// TwinCAT 3 PLC project PLC1
// ProgramVersion: 3.1.4026.22
// libraries:
//   Tc2_MC2, * (Beckhoff Automation GmbH)
//   Tc2_Standard, * (Beckhoff Automation GmbH)
//   Tc2_System, * (Beckhoff Automation GmbH)
//   Tc3_Mc3PlanarMotion, * (Beckhoff Automation GmbH)
//   Tc3_Physics, * (Beckhoff Automation GmbH)
//   Tc3_XPlanarUtility, * (Beckhoff Automation GmbH)
//   XPlanarApplication, * (Beckhoff Automation LLC)
// project tree:
//   GVLs/ GVL.TcGVL
//   / PlcTask.TcTTO
//   POUs/ MAIN.TcPOU
//   POUs/Utilities/ ErrorStep.TcPOU, NextMinorStep.TcPOU (not stored), NextStep.TcPOU (not stored)
//   POUs/XPlanarModule/ FB_XPlanarModule.TcPOU
//   POUs/XPlanarModule/StationProcesses/ FB_RotateStation.TcPOU, FB_SimulateProcess.TcPOU
// real-time tasks:
//   TASK XPlanar Task_3: cycle T#250us, priority 1, ADS port 350
//   TASK Job Task: cycle default, priority 2
//   TASK MC-Task (MET): cycle T#2ms, priority 3, ADS port 351
//   TASK MC-Task (MPT): cycle T#10ms, priority 4, ADS port 352
//   TASK PlcTask: cycle T#10ms, priority 20, ADS port 353
// variable links:
//   XPlanar MC Project/Axes/Mover4220_1 <-> TcCOM Objects/XPlanar/Mover4220_1
//     IoToMc/STD <-> OutputsToNC3/HWToNC3
//     McToIo/STD <-> InputsFromNC3/NC3ToHW
//   XPlanar MC Project/Axes/Mover4220_2 <-> TcCOM Objects/XPlanar/Mover4220_2
//     IoToMc/STD <-> OutputsToNC3/HWToNC3
//     McToIo/STD <-> InputsFromNC3/NC3ToHW
//   PLC1/PLC1 Instance <-> XPlanar MC Project/Axes/Mover4220_1
//     PlcTask Inputs/MAIN.XPlanarTable.Movers[1]._Mover.MCTOPLC/ACT <-> McToPlc/ACT
//     PlcTask Inputs/MAIN.XPlanarTable.Movers[1]._Mover.MCTOPLC/COORDMODE <-> McToPlc/COORDMODE
//     PlcTask Inputs/MAIN.XPlanarTable.Movers[1]._Mover.MCTOPLC/SET <-> McToPlc/SET
//     PlcTask Inputs/MAIN.XPlanarTable.Movers[1]._Mover.MCTOPLC/SETONTRACK <-> McToPlc/SETONTRACK
//     PlcTask Inputs/MAIN.XPlanarTable.Movers[1]._Mover.MCTOPLC/STD <-> McToPlc/STD
//     PlcTask Outputs/MAIN.XPlanarTable.Movers[1]._Mover.PLCTOMC/STD <-> PlcToMc/STD
//   PLC1/PLC1 Instance <-> XPlanar MC Project/Axes/Mover4220_2
//     PlcTask Inputs/MAIN.XPlanarTable.Movers[2]._Mover.MCTOPLC/ACT <-> McToPlc/ACT
//     PlcTask Inputs/MAIN.XPlanarTable.Movers[2]._Mover.MCTOPLC/COORDMODE <-> McToPlc/COORDMODE
//     PlcTask Inputs/MAIN.XPlanarTable.Movers[2]._Mover.MCTOPLC/SET <-> McToPlc/SET
//     PlcTask Inputs/MAIN.XPlanarTable.Movers[2]._Mover.MCTOPLC/SETONTRACK <-> McToPlc/SETONTRACK
//     PlcTask Inputs/MAIN.XPlanarTable.Movers[2]._Mover.MCTOPLC/STD <-> McToPlc/STD
//     PlcTask Outputs/MAIN.XPlanarTable.Movers[2]._Mover.PLCTOMC/STD <-> PlcToMc/STD
//   PLC1/PLC1 Instance <-> XPlanar MC Project/Groups/Environment
//     PlcTask Inputs/XPlanar.Environment.MCTOPLC_STD <-> McToPlc/STD
//   PLC1/PLC1 Instance <-> XPlanar MC Project/Groups/Track1
//     PlcTask Inputs/MAIN.XPlanarTable.Tracks[1]._Track.MCTOPLC_STD <-> McToPlc/STD
//   PLC1/PLC1 Instance <-> XPlanar MC Project/Groups/Track2
//     PlcTask Inputs/MAIN.XPlanarTable.Tracks[2]._Track.MCTOPLC_STD <-> McToPlc/STD
//   PLC1/PLC1 Instance <-> XPlanar MC Project/Groups/XPlanar
//     PlcTask Inputs/XPlanar.Group.MCTOPLC_STD <-> McToPlc/STD

CONFIGURATION PLC1
    RESOURCE PLC ON TwinCAT3
        TASK PlcTask(INTERVAL := T#10ms, PRIORITY := 20);
        PROGRAM MAIN WITH PlcTask : MAIN;
    END_RESOURCE
END_CONFIGURATION

// ---- GVLs/GVL.TcGVL
{attribute 'qualified_only'}
VAR_GLOBAL
	// Mover Velocity
	MoverVelo		: LREAL := 200;
	MoverGap		: LREAL := 180; // Do not exceed 250 mm, or go lower then default
	// Mover Rotation Velocity
	MoverSpinVelo	: LREAL := 1000;
	// Station 2 Mover Index
	Indx			: UDINT;
END_VAR

// ---- POUs/MAIN.TcPOU
PROGRAM MAIN
VAR
	XPlanarTable : FB_XPlanarModule;
	Initialize	 : BOOL; // Initialize the system
	Reset		 : BOOL; // Reset and Execute System
	Start		 : BOOL; // Run the system
	Halt		 : BOOL; // Avoid Disabling while spinning, otherwise physical sqauring of mover is required
	MachineState : (Startup,
		InitSystem,
		ResetSystem,
		Recover,
		Ready,
		Run,
		Disable);
	trig : R_TRIG;
END_VAR

//This project is a very simple "hello world" example for the APS4322 2-Tile starter kit.
//It is currently based on the XPlanarApplication library version 2.0.5 or greater.


//Keep all XPlanar motion system objects up to date every cycle
XPlanarTable.CyclicLogic();

// "Machine" Sequence
CASE MachineState OF
	Startup:	
		IF Initialize THEN
			Initialize := FALSE;
			MachineState := InitSystem;
		END_IF
	
	InitSystem:	
		IF XPlanarTable.Initialize() THEN
			MachineState := ResetSystem;
		END_IF
	
	ResetSystem:	
		IF Reset AND_THEN XPlanarTable.Reset() THEN
			Reset := FALSE;
			MachineState := Recover;
		END_IF
	
	Recover:	
		IF XPlanarTable.Recovery() THEN
			MachineState := Ready;
		END_IF
		
	Ready:
		IF Start THEN
			MachineState := Run;
		END_IF
	
	Run: 
		XPlanarTable.Execute();
	
	Disable:	
		IF XPlanarTable.Disable() THEN
			MachineState := 0;
		END_IF
END_CASE

IF Halt OR trig.Q THEN
	MachineState := Disable;
	Halt := FALSE;
END_IF

END_PROGRAM

// ---- POUs/XPlanarModule/FB_XPlanarModule.TcPOU
FUNCTION_BLOCK FB_XPlanarModule
VAR CONSTANT
	MoverCount	 : UDINT := 2;
	TrackCount	 : UDINT := 2;
	StationCount : UDINT := 2;
END_VAR

VAR
	XPlanarSystem	: FB_Component_XPlanar;
	Movers			: ARRAY[1..MoverCount] OF FB_XPlanarMover;
	Tracks			: ARRAY[1..TrackCount] OF FB_XPlanarTrackSegment;
	Stations		: ARRAY[1..StationCount] OF FB_XPlanarStationBase;
	Station1Process : FB_SimulateProcess;  //Custom process FB that can be assigned to a station
	Station2Process : FB_RotateStation;
	InitState		: (CheckForXPlanarInit, UpdateDynamics, SetStationParameters, Initialized);
END_VAR

METHOD CyclicLogic : BOOL
VAR
	i : UDINT;
END_VAR
VAR_INST
	TaskResult	: I_PlanarTaskResult;
END_VAR
XPlanarSystem.CyclicLogic();
IF NOT XPlanarSystem.Initialized THEN
	RETURN;
END_IF

//Add any logic that needs to be called every cycle here
END_METHOD

METHOD Disable : BOOL
VAR_INST
	CommandResult	: I_PlanarTaskResult;
END_VAR
CommandResult := XPlanarSystem.Abort(); // Stop Motion and Disable All Movers
IF CommandResult.Done THEN
	Disable := TRUE;
END_IF
END_METHOD

METHOD Execute : BOOL
VAR
	i : UDINT;
END_VAR
//System is 'running' cycle thru all of the stations
FOR i := 1 TO XPlanar.StationCount DO
	ip.Stations[i].Execute();
END_FOR
END_METHOD

METHOD Initialize : BOOL
VAR_INST
	i			: UDINT;
END_VAR
CASE InitState OF
	CheckForXPlanarInit: // Init Vars
		Initialize := FALSE;
		
		//Make sure the XPlanar motion system has initialized
		IF XPlanarSystem.Initialized THEN
			InitState := UpdateDynamics;
		END_IF

	UpdateDynamics: 
		//Assign Initial Application Mover Dynamics
		FOR i := 1 TO XPlanar.MoverCount DO
			ip.Movers[i].Gap						:= 200;
			ip.Movers[i].Dynamics.Movement.Velocity := GVL.MoverVelo;
			ip.Movers[i].Dynamics.Movement.Accel	:= GVL.MoverVelo * 10;
			ip.Movers[i].Dynamics.Movement.Decel	:= GVL.MoverVelo * 10;
			ip.Movers[i].Dynamics.Movement.Jerk		:= GVL.MoverVelo * 100;
			ip.Movers[i].Dynamics.Rotation.Velocity := GVL.MoverSpinVelo;
			ip.Movers[i].Dynamics.Rotation.Accel	:= GVL.MoverSpinVelo * 10;
			ip.Movers[i].Dynamics.Rotation.Decel	:= GVL.MoverSpinVelo * 10;
			ip.Movers[i].Dynamics.Rotation.Jerk		:= GVL.MoverSpinVelo * 100;
		END_FOR

		InitState := SetStationParameters;

	SetStationParameters:
		IF SetupStations() THEN
			InitState := Initialized;
		END_IF

	Initialized: // Init Complete
		Initialize := TRUE;
END_CASE
END_METHOD

METHOD Recovery : BOOL
VAR_INST
	nState			: UDINT;
	ipResult		: ARRAY[1..MoverCount] OF I_PlanarTaskResult;
	ErrorMoverId, i : UDINT;
	ItemsOk			: BOOL;
END_VAR
//This is an example of some very simple mover recovery.  
//What needs to be done to recover will be unique for each application.

CASE nState OF
	0: // Init Vars
		Recovery := FALSE;
		i := 1;
		NextStep(nState);
		
	10: // All Movers Join rack closest to their current location
		IF i <= XPlanar.MoverCount THEN
			ipResult[i] := ip.Movers[i].MoveCommand.JoinClosestTrack(FALSE);
			IF ipResult[i].Done THEN
				NextMinorStep(nState);
			ELSIF ipResult[i].Error THEN
				ErrorStep(nState);
			END_IF
		ELSE
			i := 1;
			NextStep(nState);
		END_IF

	11: //Check Mover Count
		IF i <= XPlanar.MoverCount THEN
			i	   := i + 1;
			nState := 10;
		ELSE
			i := 1;
			NextStep(nState);
		END_IF

	20: // Sort and send Movers to Stations
		FOR i := 1 TO XPlanar.MoverCount DO
			ipResult[i] := ip.Movers[i].MoveCommand.SendToStation(ip.Stations[1]);
		END_FOR

		NextStep(nState);

	30: // Wait For Mover to Move
		ItemsOk := TRUE;
		FOR i := 1 TO XPlanar.MoverCount DO
			IF NOT ipResult[i].Busy THEN
				ItemsOk := FALSE;
			END_IF

			IF ipResult[i].Error THEN
				ErrorMoverId := i;
				ErrorStep(nState);
			END_IF
		END_FOR

		IF ItemsOk THEN
			ErrorMoverId := 0;
			NextStep(nState);
		END_IF

	40: // Complete
		nState		 := 0;
		ErrorMoverId := 0;
		Recovery	 := TRUE;
END_CASE
END_METHOD

METHOD Reset : BOOL
VAR_INST
	nState		  : UDINT;
	i			  : UDINT;
	ResetOk		  : BOOL;
	ResetError	  : BOOL;
	CommandResult : I_PlanarTaskResult;
END_VAR
CASE nState OF
	0: // Init Vars
		Reset := FALSE;
		NextStep(nState);

	10: // Reset Table 
		IF XPlanarSystem.Reset().Done THEN
			NextStep(nState);
		END_IF

	20: // Reset Stations
		FOR i := 1 TO StationCount DO
			ip.Stations[i].Reset();
		END_FOR

		NextStep(nState);

	30: // Enable Movers
		CommandResult := XPlanarSystem.EnableMovers();
		IF CommandResult.Done THEN
			NextStep(nState);
		ELSIF CommandResult.Error THEN
			ErrorStep(nState);
		END_IF

	40: // Add Movers To Group
		CommandResult := XPlanarSystem.AddMoversToGroup();
		IF CommandResult.Done THEN
			NextStep(nState);
		ELSIF CommandResult.Error THEN
			ErrorStep(nState);
		END_IF

	50: // Enable Tracks
		CommandResult := XPlanarSystem.EnableTracks();
		IF CommandResult.Done THEN
			NextStep(nState);
		ELSIF CommandResult.Error THEN
			ErrorStep(nState);
		END_IF

	60: // Add Tracks To Group
		CommandResult := XPlanarSystem.AddTracksToGroup();
		IF CommandResult.Done THEN
			NextStep(nState);
		ELSIF CommandResult.Error THEN
			ErrorStep(nState);
		END_IF

	70: // Enable Group
		CommandResult := XPlanarSystem.EnableGroup();
		IF CommandResult.Done THEN
			NextStep(nState);
		ELSIF CommandResult.Error THEN
			ErrorStep(nState);
		END_IF

	80: // Complete
		Reset  := TRUE;
		nState := 0;
END_CASE
END_METHOD

METHOD PRIVATE SetupStations : BOOL
// Setup Station 1
Stations[1].ID := 1;
Stations[1].TrackID := 1;
Stations[1].Position.SetValuesXYC(120, 60, 0);
Stations[1].NextStation := ip.Stations[2];
Stations[1].Process := Station1Process; //Assign a custom process to the station
Station1Process.ProcessTime := 1.5;


// Setup Station 2
Stations[2].ID := 2;
Stations[2].TrackID := 2;
Stations[2].Position.SetValuesXYC(120, 360, 0);
Stations[2].NextStation := ip.Stations[1];
Stations[2].Process := Station2Process; //Assign a custom process to the station
Station2Process.NumberOfTurns := 2;
Station2Process.StationAngle := 0;


SetupStations:=TRUE;
END_METHOD

END_FUNCTION_BLOCK

// ---- POUs/XPlanarModule/StationProcesses/FB_SimulateProcess.TcPOU
FUNCTION_BLOCK FB_SimulateProcess IMPLEMENTS I_StationProcess
VAR
	_ProcessTime	: TIME;
END_VAR

METHOD Execute : BOOL
VAR_INPUT
	Mover	: XPlanarApplication.I_XPlanarMover;
END_VAR

VAR_INST
	SimulateTimer: TON;
END_VAR
SimulateTimer(IN := Mover <> 0, PT := _ProcessTime);
IF SimulateTimer.Q THEN
	SimulateTimer(IN := FALSE);
	Execute := TRUE;
END_IF
END_METHOD

PROPERTY ProcessTime : LREAL
SET
_ProcessTime := TO_TIME(ProcessTime * 1000);
END_SET
END_PROPERTY

END_FUNCTION_BLOCK

// ---- POUs/XPlanarModule/StationProcesses/FB_RotateStation.TcPOU
FUNCTION_BLOCK FB_RotateStation IMPLEMENTS I_StationProcess
VAR
	_StationAngle  : LREAL;
	_NumberOfTurns : DINT;

END_VAR

METHOD Execute : BOOL
VAR_INPUT
	Mover	: XPlanarApplication.I_XPlanarMover;
END_VAR

VAR_INST
	CommandResult : I_PlanarTaskResult;
END_VAR
CommandResult := Mover.MoveCommand.Rotate(_StationAngle, _NumberOfTurns);
IF CommandResult.Done THEN
	Execute := TRUE;
ELSIF CommandResult.Error THEN
	; //Command returned an error, DO SOMETHING!
END_IF
END_METHOD

PROPERTY NumberOfTurns : DINT
SET
_NumberOfTurns := NumberOfTurns;
END_SET
END_PROPERTY

PROPERTY StationAngle : LREAL
SET
_StationAngle := StationAngle;
END_SET
END_PROPERTY

END_FUNCTION_BLOCK

// ---- POUs/Utilities/ErrorStep.TcPOU
FUNCTION ErrorStep : UDINT
VAR_IN_OUT
	StateVar : UDINT;
END_VAR

ErrorStep := StateVar := ((StateVar / 10) * 10) + 9;

END_FUNCTION
